FUNCTION_BLOCK TestFB1Device
VAR_INPUT
END_VAR
VAR_OUTPUT
END_VAR
VAR
	Inst_Subdevice1:TestFB1DeviceSubdevice;
	NonPerstInt1:INT:=9;
	NonPerstInt2:INT:=10;
END_VAR
VAR PERSISTENT
	PersInt1:INT:=435;
END_VAR

NonPerstInt1:=NonPerstInt1+1;
Inst_Subdevice1();

END_FUNCTION_BLOCK

(* stored: Version 1.1.0.1, ProductVersion 3.1.4024.6
   POU TestFB1Device: Id {f43730c2-d44d-40a3-9228-071e70c60544}, SpecialFunc None *)
